// TIA Portal project "maqueta brazo" (V15)
// Vorlageprojekt für das Buch mit Zielsystem S7-1200

(* hardware
DEVICE "S7-1200-Station_1"  S7-1200 Station
   slot 0: "Baugruppenträger_0"  Rack  V1.0
   slot 1: "PLC_1"  CPU 1211C DC/DC/DC  6ES7 211-1AE40-0XB0  V4.1
*)

// ===== PLC "PLC_1"  CPU 1211C DC/DC/DC =====

VAR_GLOBAL   // PLC tag table "Standard-Variablentabelle"
   "conteo para desactivar seta" AT %MW300 : Int;
   "motor derecha" AT %Q0.4 : Bool;   // motor brazo
   "Tag_1" AT %M11.7 : Bool;
   "sensor brazo bajado_m" AT %M12.0 : Bool;
   "Step_6" AT %M12.1 : Bool;
   "conteo Z" AT %MW305 : Int;
   "Tag_2" AT %M100.5 : Bool;
   "Tag_4" AT %M150.0 : Bool;
   "conteo Y" AT %MW310 : Int;
   "brazo arriba" AT %M12.2 : Bool;
   "resto_Z" AT %MW315 : Int;
   "brazo en reposo" AT %M12.3 : Bool;
   "brazo a la derecha" AT %M12.4 : Bool;
   "brazo a la izquierda" AT %M12.5 : Bool;
   "Tag_3" AT %M106.0 : Bool;
END_VAR

VAR_GLOBAL   // PLC tag table "Tabla de variables estándar"
   "start_m" AT %M10.0 : Bool;   // Start pushbutton
   "stop_m" AT %M10.1 : Bool;   // Stop pushbutton
   "auto_man_m" AT %M10.2 : Bool;   // Auto/Manual selector
   "reset_m" AT %M10.3 : Bool;   // Reset pushbutton
   "a_0_m" AT %M10.4 : Bool;   // Eject cylinder backward
   "a_1_m" AT %M10.5 : Bool;   // Eject cylinder forward
   "b_0_m" AT %M10.6 : Bool;   // Blocking cylinder backward
   "b_1_m" AT %M10.7 : Bool;   // Blocking cylinder forward
   "Block_m" AT %M11.0 : Bool;   // Block presence
   "ALARM" AT %Q0.7 : Bool;   // Alarm lamp
   "Motor izquierda" AT %Q0.3 : Bool;   // Start conveyor / Motor brazo
   "ventosa" AT %Q0.0 : Bool;   // Eject cylinder forwards / el succionador activado
   "bajar brazo" AT %Q0.1 : Bool;   // Eject cylinder downwards / baja o sube brazo
   "B+" AT %Q0.2 : Bool;   // Blocking cylinder forwards / Este va a ser el cilindro
   "Step_0" AT %M400.0 : Bool;   // First step of grafcet
   "Step_1" AT %M400.1 : Bool;   // Feeding cylinder forwards
   "Step_2" AT %M400.2 : Bool;   // Verification cylinder downwards
   "Step_3" AT %M400.3 : Bool;   // Verification cylinder upwards
   "Step_4" AT %M400.4 : Bool;   // Feeding cylinder backwards
   "Step_5" AT %M400.5 : Bool;   // Body transfer cylinder forwards
   "ic" AT %M200.0 : Bool;   // Initial conditions
   "continue" AT %M200.1 : Bool;   // Go on with the Grafcet
   "body_ok" AT %M200.2 : Bool;   // Body in right position
   "start_stop_mode" AT %M200.3 : Bool;   // Auto / Manual mode of the station
   "no_air_pressure" AT %M200.4 : Bool;   // Station without air pressure
   "cycle" AT %M200.5 : Bool;   // Process cycle not finished
   "end_cycle" AT %M200.6 : Bool;   // Station 1 end cycle
   "FAS201_on_202" AT %Q200.0 : Bool;   // Fas-201 on for fas-202
   "FAS201_end_202" AT %Q200.1 : Bool;   // Process cycle finished at fas-201 for fas-202
   "FAS201_wrong_202" AT %Q200.2 : Bool;   // Body wrongly positioned for fas-202
   "FAS201_c1_202" AT %Q200.3 : Bool;   // Transfer cylinder forward for fas-202
   "Cell_1_ppA" AT %I200.4 : Bool;   // Palet presence fas-202
   "Cell_1_b0A" AT %I200.5 : Bool;   // Palet code bit 0 fas-202
   "Cell_1_b1A" AT %I200.6 : Bool;   // Palet code bit 1 fas-202
   "Cell_1_b2A" AT %I200.7 : Bool;   // Palet code bit 2 fas-202
   "First_SC" AT %M3.6 : Bool;
   "Tag_21" AT %M201.7 : Bool;
   "Tag_6" AT %M100.4 : Bool;
   "Cell_1_on" AT %I200.0 : Bool;   // Fas-202 on
   "Cell_1_end" AT %I200.1 : Bool;   // Cycle finished at fas-202
   "Cell_1_busy" AT %I200.2 : Bool;   // Fas-202 busy
   "Cell_1_alarm" AT %I200.3 : Bool;
   "sensor_start" AT %I1.1 : Bool;   // Capacitive sensor start conveyor
   "sensor_end" AT %I1.2 : Bool;   // Capacitive sensor end conveyor
   "brazo en movimiento" AT %I1.0 : Bool;   // Detected white block / brazo eje horizontal
   "System_Byte" AT %MB254 : Byte;
   "FirstScan" AT %M254.0 : Bool;
   "DiagStatusUpdate" AT %M254.1 : Bool;
   "AlwaysTRUE" AT %M254.2 : Bool;
   "AlwaysFALSE" AT %M254.3 : Bool;
   "start" AT %I0.2 : Bool;   // Start pushbutton
   "stop" AT %I0.1 : Bool;   // Stop pushbutton
   "auto_man" AT %I0.3 : Bool;   // Auto/Manual selector
   "reset" AT %I0.0 : Bool;   // Reset pushbutton
   "ventosa activada" AT %I0.4 : Bool;   // Eject cylinder backward / Ventosa
   "sensor pieza" AT %I0.5 : Bool;   // Eject cylinder forward / Botón para verificar si hay pieza
   "b_0" AT %I0.6 : Bool;   // Blocking cylinder backward / cilindro detrás
   "b_1" AT %I0.7 : Bool;   // Blocking cylinder forward / cilindro delante
   "Sensor brazo bajado" AT %I1.3 : Bool;   // Block presence / Sensor que indica si el brazo está bajando o subiendo
   "Sensor_start_m" AT %M11.1 : Bool;
   "sensor_end_m" AT %M11.2 : Bool;
   "brazo en movimiento _m" AT %M11.3 : Bool;
   "Pieza a la espera" AT %M11.4 : Bool;   // Se activa cuando hay una pieza en la cinta
   "pieza cogida" AT %M11.5 : Bool;   // Se activa cuando detecta que la pieza es blanca / variable que nos indica si el brazo ha cogido la pieza
   "Piezas" AT %M11.6 : Bool;   // Cuenta el número de piezas
   "reinicio" AT %M400.6 : Bool;
END_VAR

VAR_GLOBAL CONSTANT   // PLC tag table "Tabla de variables estándar"
   "Local~AI2_1" : Hw_SubModule := 264;
   "Local~DI14_DQ10_1" : Hw_SubModule := 265;
   "OB_Main(1)" : OB_PCYCLE := 1;
   "OB_Diagnostic error interrupt" : OB_DIAG := 82;
   "None" : Pip := 65535;
   "Automatic update" : Pip := 0;
   "PIP 1" : Pip := 1;
   "PIP 2" : Pip := 2;
   "PIP 3" : Pip := 3;
   "PIP 4" : Pip := 4;
   "PIP OB Servo" : Pip := 32768;
   "Local~Interfaz_PROFINET_1~IODevice" : Hw_Device := 271;
   "Local~Interfaz_PROFINET_1~Transfer_area_1" : Hw_SubModule := 273;
   "Local~Interfaz_PROFINET_1~Transfer_area_2" : Hw_SubModule := 274;
   "Local~Exec(1)" : Hw_SubModule := 52;
   "Local(1)" : Hw_SubModule := 49;
   "Local~Interfaz_PROFINET_1~Puerto_1" : Hw_Interface := 65;
   "Local~MC(1)" : Hw_SubModule := 51;
   "Local~Common(1)" : Hw_SubModule := 50;
   "Local~Device(1)" : Hw_Device := 32;
   "Local~Configuration(1)" : Hw_SubModule := 33;
   "Local~HSC_1(1)" : Hw_Hsc := 258;
   "Local~HSC_2(1)" : Hw_Hsc := 259;
   "Local~HSC_3(1)" : Hw_Hsc := 260;
   "Local~HSC_4(1)" : Hw_Hsc := 261;
   "Local~HSC_5(1)" : Hw_Hsc := 262;
   "Local~HSC_6(1)" : Hw_Hsc := 263;
   "Local~Pulse_1(1)" : Hw_Pwm := 266;
   "Local~Pulse_2(1)" : Hw_Pwm := 267;
   "Local~Pulse_3(1)" : Hw_Pwm := 269;
   "Local~Pulse_4(1)" : Hw_Pwm := 270;
   "Local~Interfaz_PROFINET_1" : Hw_Interface := 64;
   "Local~AQ_2x14BIT_1" : Hw_SubModule := 275;
   "Local~DQ_4x24VDC_1" : Hw_SubModule := 276;
   "OB_Startup" : OB_STARTUP := 100;
END_VAR

// folder: System blocks/Program resources

DATA_BLOCK "TIMER_1"   // DB1
{ S7_Optimized_Access := 'TRUE' }
AUTHOR : Simatic
FAMILY : IEC
NAME : IEC_TMR
VERSION : 1.0
// stored: InstanceOfName IEC_TIMER
"IEC_TIMER"
BEGIN
END_DATA_BLOCK

DATA_BLOCK "TIMER_2"   // DB2
{ S7_Optimized_Access := 'TRUE' }
AUTHOR : Simatic
FAMILY : IEC
NAME : IEC_TMR
VERSION : 1.0
// stored: InstanceOfName IEC_TIMER
"IEC_TIMER"
BEGIN
END_DATA_BLOCK

DATA_BLOCK "TIMER_3"   // DB3
{ S7_Optimized_Access := 'TRUE' }
AUTHOR : Simatic
FAMILY : IEC
NAME : IEC_TMR
VERSION : 1.0
// stored: InstanceOfName IEC_TIMER
"IEC_TIMER"
BEGIN
END_DATA_BLOCK

DATA_BLOCK "IEC_Counter_0_DB"   // DB4
{ S7_Optimized_Access := 'TRUE' }
AUTHOR : Simatic
FAMILY : IEC
NAME : CNTR
VERSION : 1.0
// stored: InstanceOfName IEC_COUNTER
"IEC_COUNTER"
BEGIN
END_DATA_BLOCK

DATA_BLOCK "TIMER_6"   // DB5
{ S7_Optimized_Access := 'TRUE' }
AUTHOR : Simatic
FAMILY : IEC
NAME : IEC_TMR
VERSION : 1.0
// stored: InstanceOfName IEC_TIMER
"IEC_TIMER"
BEGIN
END_DATA_BLOCK

DATA_BLOCK "TIMER_8"   // DB6
{ S7_Optimized_Access := 'TRUE' }
AUTHOR : Simatic
FAMILY : IEC
NAME : IEC_TMR
VERSION : 1.0
// stored: InstanceOfName IEC_TIMER
"IEC_TIMER"
BEGIN
END_DATA_BLOCK

DATA_BLOCK "IEC_Timer_0_DB_3"   // DB7
{ S7_Optimized_Access := 'TRUE' }
AUTHOR : Simatic
FAMILY : IEC
NAME : IEC_TMR
VERSION : 1.0
// stored: InstanceOfName IEC_TIMER
"IEC_TIMER"
BEGIN
END_DATA_BLOCK

DATA_BLOCK "IEC_Timer_0_DB"   // DB8
{ S7_Optimized_Access := 'TRUE' }
AUTHOR : Simatic
FAMILY : IEC
NAME : IEC_TMR
VERSION : 1.0
// stored: InstanceOfName IEC_TIMER
"IEC_TIMER"
BEGIN
END_DATA_BLOCK

DATA_BLOCK "IEC_Timer_0_DB_1"   // DB9
{ S7_Optimized_Access := 'TRUE' }
AUTHOR : Simatic
FAMILY : IEC
NAME : IEC_TMR
VERSION : 1.0
// stored: InstanceOfName IEC_TIMER
"IEC_TIMER"
BEGIN
END_DATA_BLOCK

DATA_BLOCK "IEC_Counter_0_DB_2"   // DB10
{ S7_Optimized_Access := 'TRUE' }
AUTHOR : Simatic
FAMILY : IEC
NAME : CNTR
VERSION : 1.0
// stored: InstanceOfName IEC_COUNTER
"IEC_COUNTER"
BEGIN
END_DATA_BLOCK

DATA_BLOCK "IEC_Timer_0_DB_4"   // DB11
{ S7_Optimized_Access := 'TRUE' }
AUTHOR : Simatic
FAMILY : IEC
NAME : IEC_TMR
VERSION : 1.0
// stored: InstanceOfName IEC_TIMER
"IEC_TIMER"
BEGIN
END_DATA_BLOCK

DATA_BLOCK "IEC_Counter_0_DB_3"   // DB12
{ S7_Optimized_Access := 'TRUE' }
AUTHOR : Simatic
FAMILY : IEC
NAME : CNTR
VERSION : 1.0
// stored: InstanceOfName IEC_COUNTER
"IEC_COUNTER"
BEGIN
END_DATA_BLOCK

DATA_BLOCK "IEC_Timer_0_DB_2"   // DB13
{ S7_Optimized_Access := 'TRUE' }
AUTHOR : Simatic
FAMILY : IEC
NAME : IEC_TMR
VERSION : 1.0
// stored: InstanceOfName IEC_TIMER
"IEC_TIMER"
BEGIN
END_DATA_BLOCK

DATA_BLOCK "IEC_Timer_0_DB_5"   // DB14
{ S7_Optimized_Access := 'TRUE' }
AUTHOR : Simatic
FAMILY : IEC
NAME : IEC_TMR
VERSION : 1.0
// stored: InstanceOfName IEC_TIMER
"IEC_TIMER"
BEGIN
END_DATA_BLOCK

DATA_BLOCK "IEC_Timer_0_DB_7"   // DB16
{ S7_Optimized_Access := 'TRUE' }
AUTHOR : Simatic
FAMILY : IEC
NAME : IEC_TMR
VERSION : 1.0
// stored: InstanceOfName IEC_TIMER
"IEC_TIMER"
BEGIN
END_DATA_BLOCK

// folder: (top level)

FUNCTION "STEPS" : Void   // FC1, LAD
TITLE = STEPS
{ S7_Optimized_Access := 'TRUE' }
VERSION : 0.1
   VAR_TEMP   // added for the SCL form of the ladder/FBD networks
      _w1 : Bool;
   END_VAR
BEGIN

REGION Network 1: STEP 0 / Reposo
   // FIRST STEP OF GRAFCET / Para entrar a este estado, el brazo ha de estar en su posición inicial, con el brazo arriba y en posición de reposo.
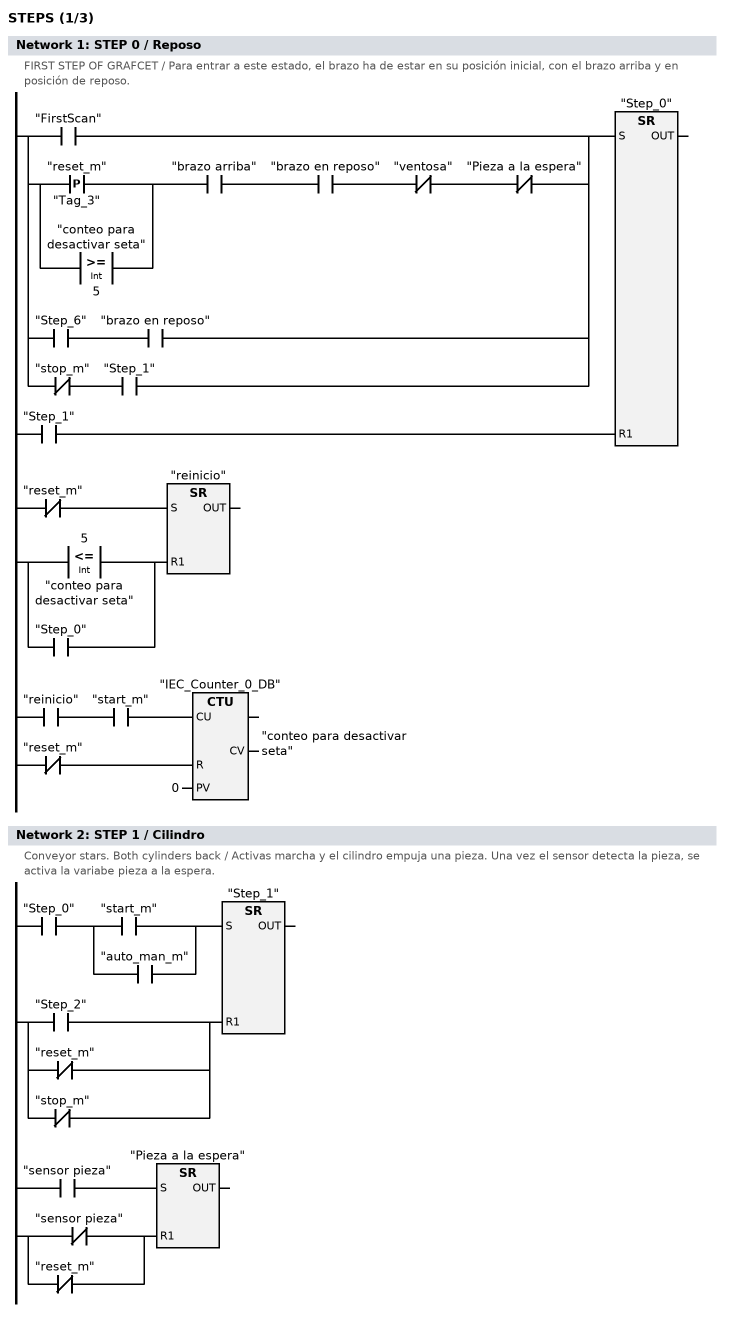
   #_w1 := "reset_m" AND NOT "Tag_3";   // rising edge of "reset_m"
   "Tag_3" := "reset_m";
   IF "FirstScan" OR ((#_w1 OR ("conteo para desactivar seta" >= 5)) AND "brazo arriba" AND "brazo en reposo" AND NOT "ventosa" AND NOT "Pieza a la espera") OR ("Step_6" AND "brazo en reposo") OR (NOT "stop_m" AND "Step_1") THEN
       "Step_0" := TRUE;   // SR flip-flop
   END_IF;
   IF "Step_1" THEN "Step_0" := FALSE; END_IF;
   IF NOT "reset_m" THEN
       "reinicio" := TRUE;   // SR flip-flop
   END_IF;
   IF (5 <= "conteo para desactivar seta") OR "Step_0" THEN "reinicio" := FALSE; END_IF;
   "IEC_Counter_0_DB".CTU(CU := "reinicio" AND "start_m",
                          R := NOT "reset_m",
                          PV := 0,
                          CV => "conteo para desactivar seta");
END_REGION

REGION Network 2: STEP 1 / Cilindro
   // Conveyor stars. Both cylinders back / Activas marcha y el cilindro empuja una pieza. Una vez el sensor detecta la pieza, se activa la variabe pieza a la espera.
   RUNG wire#powerrail
      Contact( "Step_0" )
      wire#w1
      Contact( "start_m" )
      wire#w2
      S_SR(operand := "Step_1", r1 := wire#w3)
   END_RUNG
   RUNG wire#w1
      Contact( "auto_man_m" )
   END_RUNG wire#w2
   RUNG wire#powerrail
      Contact( "Step_2" )
   END_RUNG wire#w3
   RUNG wire#powerrail
      I_Contact( "reset_m" )
   END_RUNG wire#w3
   RUNG wire#powerrail
      I_Contact( "stop_m" )
   END_RUNG wire#w3
   RUNG wire#powerrail
      Contact( "sensor pieza" )
      S_SR(operand := "Pieza a la espera", r1 := wire#w4)
   END_RUNG
   RUNG wire#powerrail
      I_Contact( "sensor pieza" )
   END_RUNG wire#w4
   RUNG wire#powerrail
      I_Contact( "reset_m" )
   END_RUNG wire#w4
   // the same network as SCL:
   IF "Step_0" AND ("start_m" OR "auto_man_m") THEN
       "Step_1" := TRUE;   // SR flip-flop
   END_IF;
   IF "Step_2" OR NOT "reset_m" OR NOT "stop_m" THEN "Step_1" := FALSE; END_IF;
   IF "sensor pieza" THEN
       "Pieza a la espera" := TRUE;   // SR flip-flop
   END_IF;
   IF NOT "sensor pieza" OR NOT "reset_m" THEN "Pieza a la espera" := FALSE; END_IF;
END_REGION

REGION Network 3: STEP 2 / movimiento brazo
   // Block the body / una vez detectado que hay pieza, el brazo deja su posición de reposo y hace un movimiento a la derecha para posicionarse encima de la pieza.
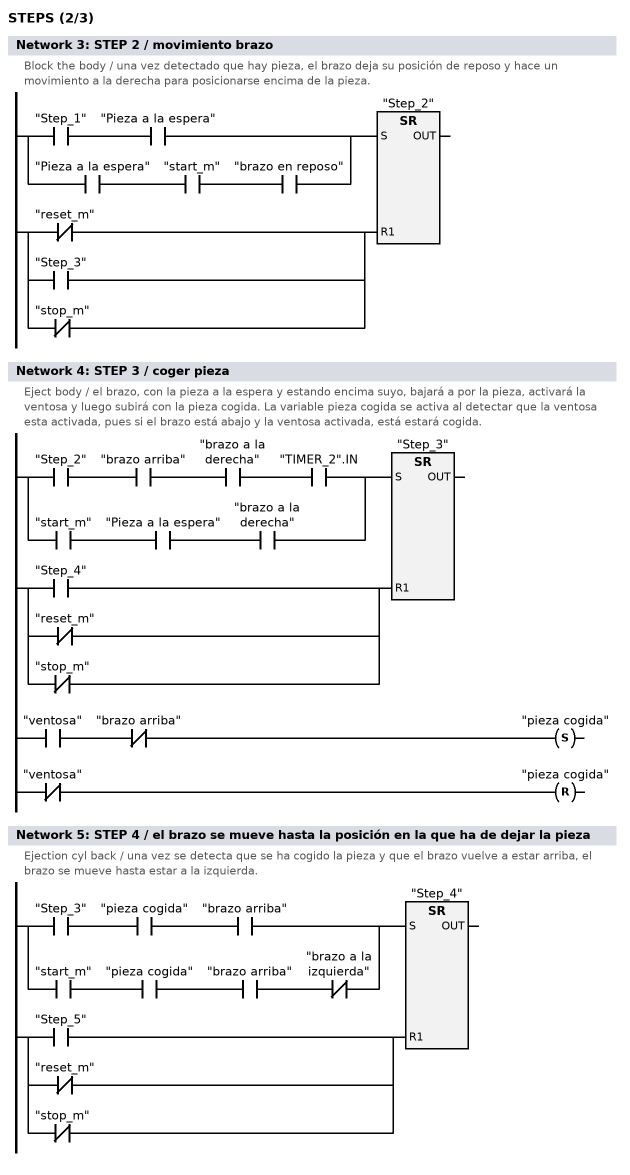
   RUNG wire#powerrail
      Contact( "Step_1" )
      Contact( "Pieza a la espera" )
      wire#w1
      S_SR(operand := "Step_2", r1 := wire#w2)
   END_RUNG
   RUNG wire#powerrail
      Contact( "Pieza a la espera" )
      Contact( "start_m" )
      Contact( "brazo en reposo" )
   END_RUNG wire#w1
   RUNG wire#powerrail
      I_Contact( "reset_m" )
   END_RUNG wire#w2
   RUNG wire#powerrail
      Contact( "Step_3" )
   END_RUNG wire#w2
   RUNG wire#powerrail
      I_Contact( "stop_m" )
   END_RUNG wire#w2
   // the same network as SCL:
   IF ("Step_1" AND "Pieza a la espera") OR ("Pieza a la espera" AND "start_m" AND "brazo en reposo") THEN
       "Step_2" := TRUE;   // SR flip-flop
   END_IF;
   IF NOT "reset_m" OR "Step_3" OR NOT "stop_m" THEN "Step_2" := FALSE; END_IF;
END_REGION

REGION Network 4: STEP 3 / coger pieza
   // Eject body / el brazo, con la pieza a la espera y estando encima suyo, bajará a por la pieza, activará la ventosa y luego subirá con la pieza cogida. La variable pieza cogida se activa al detectar que la ventosa esta activada, pues si el brazo está abajo y la ventosa activada, está estará cogida.
   RUNG wire#powerrail
      Contact( "Step_2" )
      Contact( "brazo arriba" )
      Contact( "brazo a la derecha" )
      Contact( "TIMER_2".IN )
      wire#w1
      S_SR(operand := "Step_3", r1 := wire#w2)
   END_RUNG
   RUNG wire#powerrail
      Contact( "start_m" )
      Contact( "Pieza a la espera" )
      Contact( "brazo a la derecha" )
   END_RUNG wire#w1
   RUNG wire#powerrail
      Contact( "Step_4" )
   END_RUNG wire#w2
   RUNG wire#powerrail
      I_Contact( "reset_m" )
   END_RUNG wire#w2
   RUNG wire#powerrail
      I_Contact( "stop_m" )
   END_RUNG wire#w2
   RUNG wire#powerrail
      Contact( "ventosa" )
      I_Contact( "brazo arriba" )
      S_Coil( "pieza cogida" )
   END_RUNG
   RUNG wire#powerrail
      I_Contact( "ventosa" )
      R_Coil( "pieza cogida" )
   END_RUNG
   // the same network as SCL:
   IF ("Step_2" AND "brazo arriba" AND "brazo a la derecha" AND "TIMER_2".IN) OR ("start_m" AND "Pieza a la espera" AND "brazo a la derecha") THEN
       "Step_3" := TRUE;   // SR flip-flop
   END_IF;
   IF "Step_4" OR NOT "reset_m" OR NOT "stop_m" THEN "Step_3" := FALSE; END_IF;
   IF "ventosa" AND NOT "brazo arriba" THEN "pieza cogida" := TRUE; END_IF;
   IF NOT "ventosa" THEN "pieza cogida" := FALSE; END_IF;
END_REGION

REGION Network 5: STEP 4 / el brazo se mueve hasta la posición en la que ha de dejar la pieza
   // Ejection cyl back / una vez se detecta que se ha cogido la pieza y que el brazo vuelve a estar arriba, el brazo se mueve hasta estar a la izquierda.
   RUNG wire#powerrail
      Contact( "Step_3" )
      Contact( "pieza cogida" )
      Contact( "brazo arriba" )
      wire#w1
      S_SR(operand := "Step_4", r1 := wire#w2)
   END_RUNG
   RUNG wire#powerrail
      Contact( "start_m" )
      Contact( "pieza cogida" )
      Contact( "brazo arriba" )
      I_Contact( "brazo a la izquierda" )
   END_RUNG wire#w1
   RUNG wire#powerrail
      Contact( "Step_5" )
   END_RUNG wire#w2
   RUNG wire#powerrail
      I_Contact( "reset_m" )
   END_RUNG wire#w2
   RUNG wire#powerrail
      I_Contact( "stop_m" )
   END_RUNG wire#w2
   // the same network as SCL:
   IF ("Step_3" AND "pieza cogida" AND "brazo arriba") OR ("start_m" AND "pieza cogida" AND "brazo arriba" AND NOT "brazo a la izquierda") THEN
       "Step_4" := TRUE;   // SR flip-flop
   END_IF;
   IF "Step_5" OR NOT "reset_m" OR NOT "stop_m" THEN "Step_4" := FALSE; END_IF;
END_REGION

REGION Network 6: dejar pieza
   // una vez detecta que la pieza está a la izquierda, con la pieza cogida, bajará el brazo para dejar la pieza.
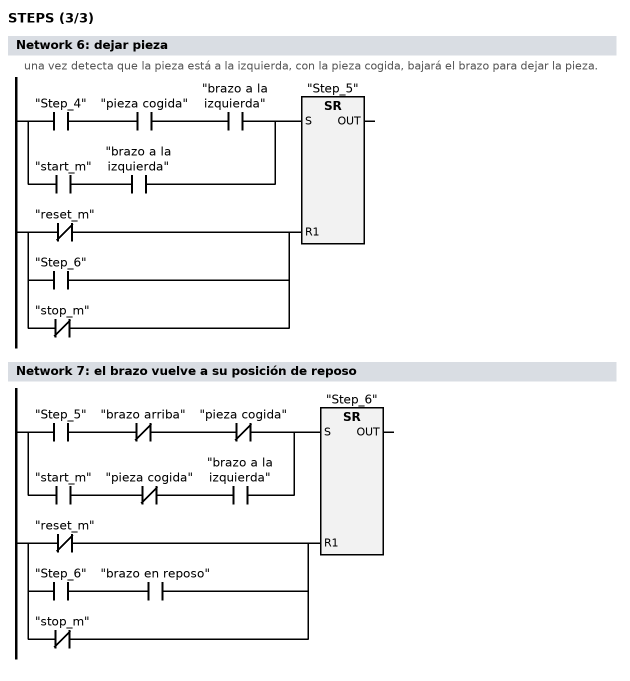
   RUNG wire#powerrail
      Contact( "Step_4" )
      Contact( "pieza cogida" )
      Contact( "brazo a la izquierda" )
      wire#w1
      S_SR(operand := "Step_5", r1 := wire#w2)
   END_RUNG
   RUNG wire#powerrail
      Contact( "start_m" )
      Contact( "brazo a la izquierda" )
   END_RUNG wire#w1
   RUNG wire#powerrail
      I_Contact( "reset_m" )
   END_RUNG wire#w2
   RUNG wire#powerrail
      Contact( "Step_6" )
   END_RUNG wire#w2
   RUNG wire#powerrail
      I_Contact( "stop_m" )
   END_RUNG wire#w2
   // the same network as SCL:
   IF ("Step_4" AND "pieza cogida" AND "brazo a la izquierda") OR ("start_m" AND "brazo a la izquierda") THEN
       "Step_5" := TRUE;   // SR flip-flop
   END_IF;
   IF NOT "reset_m" OR "Step_6" OR NOT "stop_m" THEN "Step_5" := FALSE; END_IF;
END_REGION

REGION Network 7: el brazo vuelve a su posición de reposo
   RUNG wire#powerrail
      Contact( "Step_5" )
      I_Contact( "brazo arriba" )
      I_Contact( "pieza cogida" )
      wire#w1
      S_SR(operand := "Step_6", r1 := wire#w2)
   END_RUNG
   RUNG wire#powerrail
      Contact( "start_m" )
      I_Contact( "pieza cogida" )
      Contact( "brazo a la izquierda" )
   END_RUNG wire#w1
   RUNG wire#powerrail
      I_Contact( "reset_m" )
   END_RUNG wire#w2
   RUNG wire#powerrail
      Contact( "Step_6" )
      Contact( "brazo en reposo" )
   END_RUNG wire#w2
   RUNG wire#powerrail
      I_Contact( "stop_m" )
   END_RUNG wire#w2
   // the same network as SCL:
   #_w1 := NOT "reset_m" OR ("Step_6" AND "brazo en reposo") OR NOT "stop_m";
   IF ("Step_5" AND NOT "brazo arriba" AND NOT "pieza cogida") OR ("start_m" AND NOT "pieza cogida" AND "brazo a la izquierda") THEN
       "Step_6" := TRUE;   // SR flip-flop
   END_IF;
   IF #_w1 THEN "Step_6" := FALSE; END_IF;
END_REGION
END_FUNCTION

FUNCTION "TIMERS" : Void   // FC2, LAD
TITLE = TIMERS
{ S7_Optimized_Access := 'TRUE' }
VERSION : 0.1
BEGIN

REGION Network 1: TIMER 1
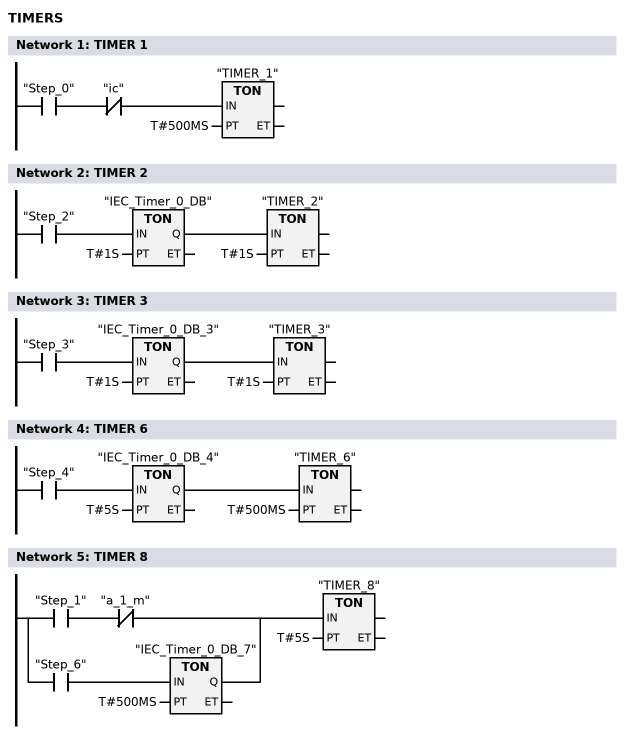
   "TIMER_1".TON(IN := "Step_0" AND NOT "ic", PT := T#500MS);
END_REGION

REGION Network 2: TIMER 2
   "IEC_Timer_0_DB".TON(IN := "Step_2", PT := T#1S);
   "TIMER_2".TON(IN := "IEC_Timer_0_DB".Q, PT := T#1S);
END_REGION

REGION Network 3: TIMER 3
   "IEC_Timer_0_DB_3".TON(IN := "Step_3", PT := T#1S);
   "TIMER_3".TON(IN := "IEC_Timer_0_DB_3".Q, PT := T#1S);
END_REGION

REGION Network 4: TIMER 6
   "IEC_Timer_0_DB_4".TON(IN := "Step_4", PT := T#5S);
   "TIMER_6".TON(IN := "IEC_Timer_0_DB_4".Q, PT := T#500MS);
END_REGION

REGION Network 5: TIMER 8
   "IEC_Timer_0_DB_7".TON(IN := "Step_6", PT := T#500MS);
   "TIMER_8".TON(IN := ("Step_1" AND NOT "a_1_m") OR "IEC_Timer_0_DB_7".Q, PT := T#5S);
END_REGION
END_FUNCTION

FUNCTION "WORKBITS" : Void   // FC3, LAD
TITLE = WORKBITS
{ S7_Optimized_Access := 'TRUE' }
VERSION : 0.1
BEGIN

REGION Network 1: START STOP MODE
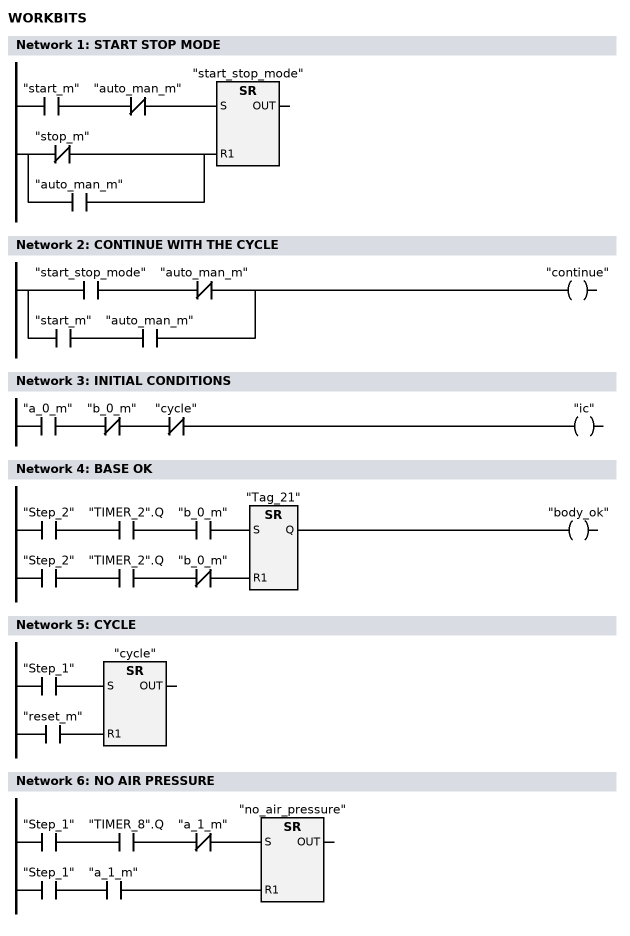
   RUNG wire#powerrail
      Contact( "start_m" )
      I_Contact( "auto_man_m" )
      S_SR(operand := "start_stop_mode", r1 := wire#w1)
   END_RUNG
   RUNG wire#powerrail
      I_Contact( "stop_m" )
   END_RUNG wire#w1
   RUNG wire#powerrail
      Contact( "auto_man_m" )
   END_RUNG wire#w1
   // the same network as SCL:
   IF "start_m" AND NOT "auto_man_m" THEN
       "start_stop_mode" := TRUE;   // SR flip-flop
   END_IF;
   IF NOT "stop_m" OR "auto_man_m" THEN "start_stop_mode" := FALSE; END_IF;
END_REGION

REGION Network 2: CONTINUE WITH THE CYCLE
   RUNG wire#powerrail
      Contact( "start_stop_mode" )
      I_Contact( "auto_man_m" )
      wire#w1
      Coil( "continue" )
   END_RUNG
   RUNG wire#powerrail
      Contact( "start_m" )
      Contact( "auto_man_m" )
   END_RUNG wire#w1
   // the same network as SCL:
   "continue" := ("start_stop_mode" AND NOT "auto_man_m") OR ("start_m" AND "auto_man_m");
END_REGION

REGION Network 3: INITIAL CONDITIONS
   RUNG wire#powerrail
      Contact( "a_0_m" )
      I_Contact( "b_0_m" )
      I_Contact( "cycle" )
      Coil( "ic" )
   END_RUNG
   // the same network as SCL:
   "ic" := "a_0_m" AND NOT "b_0_m" AND NOT "cycle";
END_REGION

REGION Network 4: BASE OK
   RUNG wire#powerrail
      Contact( "Step_2" )
      Contact( "TIMER_2".Q )
      Contact( "b_0_m" )
      S_SR(operand := "Tag_21", r1 := wire#w1)
      Coil( "body_ok" )
   END_RUNG
   RUNG wire#powerrail
      Contact( "Step_2" )
      Contact( "TIMER_2".Q )
      I_Contact( "b_0_m" )
   END_RUNG wire#w1
   // the same network as SCL:
   IF "Step_2" AND "TIMER_2".Q AND "b_0_m" THEN
       "Tag_21" := TRUE;   // SR flip-flop
   END_IF;
   IF "Step_2" AND "TIMER_2".Q AND NOT "b_0_m" THEN "Tag_21" := FALSE; END_IF;
   "body_ok" := "Tag_21";
END_REGION

REGION Network 5: CYCLE
   RUNG wire#powerrail
      Contact( "Step_1" )
      S_SR(operand := "cycle", r1 := wire#w1)
   END_RUNG
   RUNG wire#powerrail
      Contact( "reset_m" )
   END_RUNG wire#w1
   // the same network as SCL:
   IF "Step_1" THEN
       "cycle" := TRUE;   // SR flip-flop
   END_IF;
   IF "reset_m" THEN "cycle" := FALSE; END_IF;
END_REGION

REGION Network 6: NO AIR PRESSURE
   RUNG wire#powerrail
      Contact( "Step_1" )
      Contact( "TIMER_8".Q )
      I_Contact( "a_1_m" )
      S_SR(operand := "no_air_pressure", r1 := wire#w1)
   END_RUNG
   RUNG wire#powerrail
      Contact( "Step_1" )
      Contact( "a_1_m" )
   END_RUNG wire#w1
   // the same network as SCL:
   IF "Step_1" AND "TIMER_8".Q AND NOT "a_1_m" THEN
       "no_air_pressure" := TRUE;   // SR flip-flop
   END_IF;
   IF "Step_1" AND "a_1_m" THEN "no_air_pressure" := FALSE; END_IF;
END_REGION
END_FUNCTION

FUNCTION "OUTPUTS" : Void   // FC4, LAD
TITLE = OUTPUTS
{ S7_Optimized_Access := 'TRUE' }
VERSION : 0.1
BEGIN

REGION Network 1: ALARM
   // NO MATERIAL LAMP FLASHING
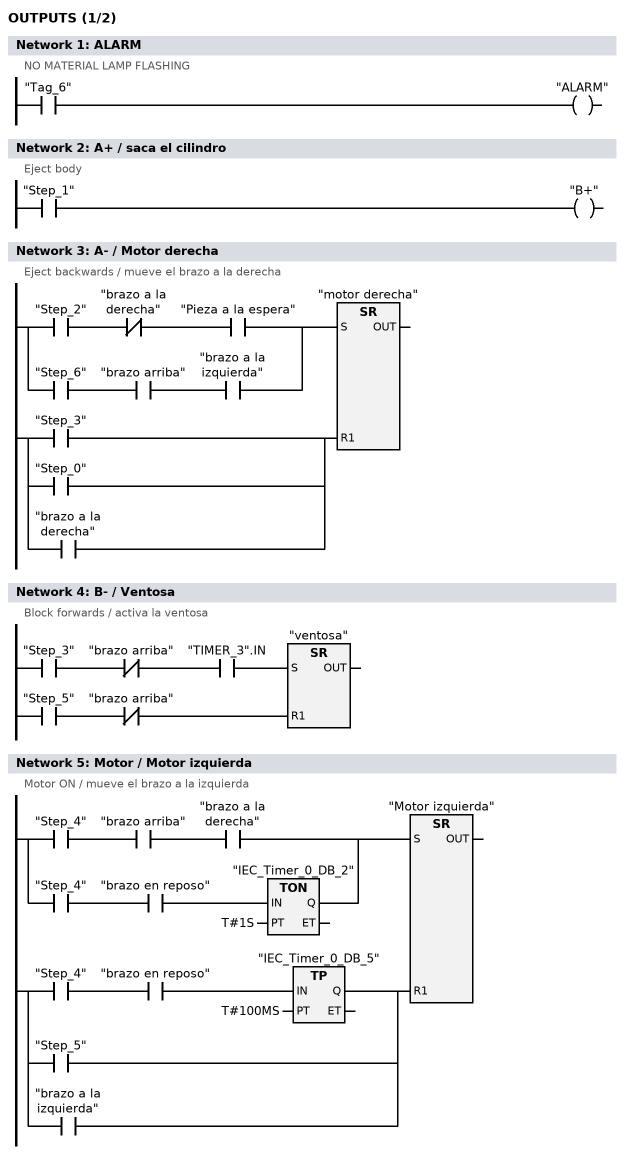
   RUNG wire#powerrail
      Contact( "Tag_6" )
      Coil( "ALARM" )
   END_RUNG
   // the same network as SCL:
   "ALARM" := "Tag_6";
END_REGION

REGION Network 2: A+ / saca el cilindro
   // Eject body
   RUNG wire#powerrail
      Contact( "Step_1" )
      Coil( "B+" )
   END_RUNG
   // the same network as SCL:
   "B+" := "Step_1";
END_REGION

REGION Network 3: A- / Motor derecha
   // Eject backwards / mueve el brazo a la derecha
   RUNG wire#powerrail
      Contact( "Step_2" )
      I_Contact( "brazo a la derecha" )
      Contact( "Pieza a la espera" )
      wire#w1
      S_SR(operand := "motor derecha", r1 := wire#w2)
   END_RUNG
   RUNG wire#powerrail
      Contact( "Step_6" )
      Contact( "brazo arriba" )
      Contact( "brazo a la izquierda" )
   END_RUNG wire#w1
   RUNG wire#powerrail
      Contact( "Step_3" )
   END_RUNG wire#w2
   RUNG wire#powerrail
      Contact( "Step_0" )
   END_RUNG wire#w2
   RUNG wire#powerrail
      Contact( "brazo a la derecha" )
   END_RUNG wire#w2
   // the same network as SCL:
   IF ("Step_2" AND NOT "brazo a la derecha" AND "Pieza a la espera") OR ("Step_6" AND "brazo arriba" AND "brazo a la izquierda") THEN
       "motor derecha" := TRUE;   // SR flip-flop
   END_IF;
   IF "Step_3" OR "Step_0" OR "brazo a la derecha" THEN "motor derecha" := FALSE; END_IF;
END_REGION

REGION Network 4: B- / Ventosa
   // Block forwards / activa la ventosa
   RUNG wire#powerrail
      Contact( "Step_3" )
      I_Contact( "brazo arriba" )
      Contact( "TIMER_3".IN )
      S_SR(operand := "ventosa", r1 := wire#w1)
   END_RUNG
   RUNG wire#powerrail
      Contact( "Step_5" )
      I_Contact( "brazo arriba" )
   END_RUNG wire#w1
   // the same network as SCL:
   IF "Step_3" AND NOT "brazo arriba" AND "TIMER_3".IN THEN
       "ventosa" := TRUE;   // SR flip-flop
   END_IF;
   IF "Step_5" AND NOT "brazo arriba" THEN "ventosa" := FALSE; END_IF;
END_REGION

REGION Network 5: Motor / Motor izquierda
   // Motor ON / mueve el brazo a la izquierda
   "IEC_Timer_0_DB_2".TON(IN := "Step_4" AND "brazo en reposo", PT := T#1S);
   "IEC_Timer_0_DB_5".TP(IN := "Step_4" AND "brazo en reposo", PT := T#100MS);
   IF ("Step_4" AND "brazo arriba" AND "brazo a la derecha") OR "IEC_Timer_0_DB_2".Q THEN
       "Motor izquierda" := TRUE;   // SR flip-flop
   END_IF;
   IF "IEC_Timer_0_DB_5".Q OR "Step_5" OR "brazo a la izquierda" THEN "Motor izquierda" := FALSE; END_IF;
END_REGION

REGION Network 6: bajar-subir brazo
   // baja el brazo
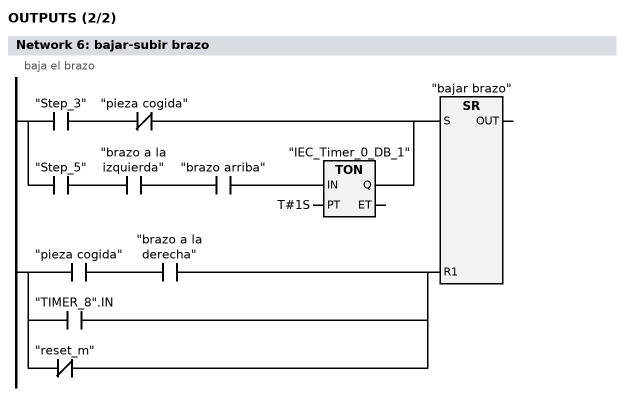
   "IEC_Timer_0_DB_1".TON(IN := "Step_5" AND "brazo a la izquierda" AND "brazo arriba", PT := T#1S);
   IF ("Step_3" AND NOT "pieza cogida") OR "IEC_Timer_0_DB_1".Q THEN
       "bajar brazo" := TRUE;   // SR flip-flop
   END_IF;
   IF ("pieza cogida" AND "brazo a la derecha") OR "TIMER_8".IN OR NOT "reset_m" THEN
       "bajar brazo" := FALSE;
   END_IF;
END_REGION
END_FUNCTION

FUNCTION "COMMS" : Void   // FC5, LAD
TITLE = PROFINET COMMUNICATION
{ S7_Optimized_Access := 'TRUE' }
VERSION : 0.1
BEGIN

REGION Network 1: FAS-201 ON FOR FAS-202
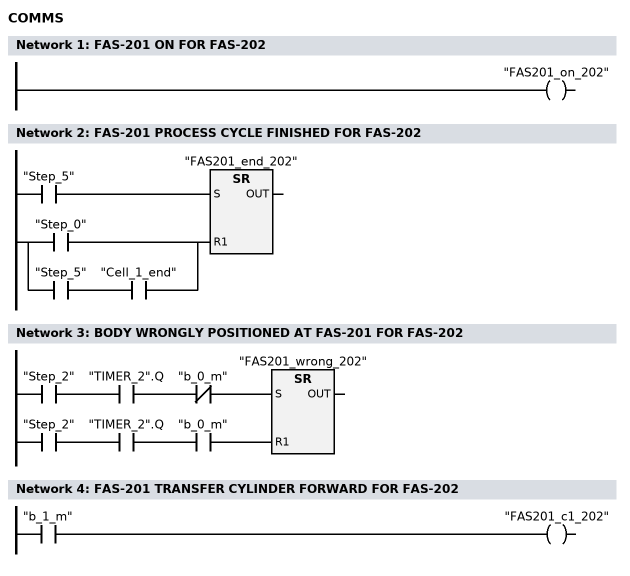
   RUNG wire#powerrail
      Coil( "FAS201_on_202" )
   END_RUNG
   // the same network as SCL:
   "FAS201_on_202" := TRUE;
END_REGION

REGION Network 2: FAS-201 PROCESS CYCLE FINISHED FOR FAS-202
   RUNG wire#powerrail
      Contact( "Step_5" )
      S_SR(operand := "FAS201_end_202", r1 := wire#w1)
   END_RUNG
   RUNG wire#powerrail
      Contact( "Step_0" )
   END_RUNG wire#w1
   RUNG wire#powerrail
      Contact( "Step_5" )
      Contact( "Cell_1_end" )
   END_RUNG wire#w1
   // the same network as SCL:
   IF "Step_5" THEN
       "FAS201_end_202" := TRUE;   // SR flip-flop
   END_IF;
   IF "Step_0" OR ("Step_5" AND "Cell_1_end") THEN "FAS201_end_202" := FALSE; END_IF;
END_REGION

REGION Network 3: BODY WRONGLY POSITIONED AT FAS-201 FOR FAS-202
   RUNG wire#powerrail
      Contact( "Step_2" )
      Contact( "TIMER_2".Q )
      I_Contact( "b_0_m" )
      S_SR(operand := "FAS201_wrong_202", r1 := wire#w1)
   END_RUNG
   RUNG wire#powerrail
      Contact( "Step_2" )
      Contact( "TIMER_2".Q )
      Contact( "b_0_m" )
   END_RUNG wire#w1
   // the same network as SCL:
   IF "Step_2" AND "TIMER_2".Q AND NOT "b_0_m" THEN
       "FAS201_wrong_202" := TRUE;   // SR flip-flop
   END_IF;
   IF "Step_2" AND "TIMER_2".Q AND "b_0_m" THEN "FAS201_wrong_202" := FALSE; END_IF;
END_REGION

REGION Network 4: FAS-201 TRANSFER CYLINDER FORWARD FOR FAS-202
   RUNG wire#powerrail
      Contact( "b_1_m" )
      Coil( "FAS201_c1_202" )
   END_RUNG
   // the same network as SCL:
   "FAS201_c1_202" := "b_1_m";
END_REGION
END_FUNCTION

FUNCTION "I_to_M" : Void   // FC6, LAD
{ S7_Optimized_Access := 'TRUE' }
VERSION : 0.1
BEGIN

REGION Network 1: Entradas Byte 0
   // El byte 0 de entradas asigna las marcas del byte 0 los a0-1 y b0-1 son las entradas de cilindro
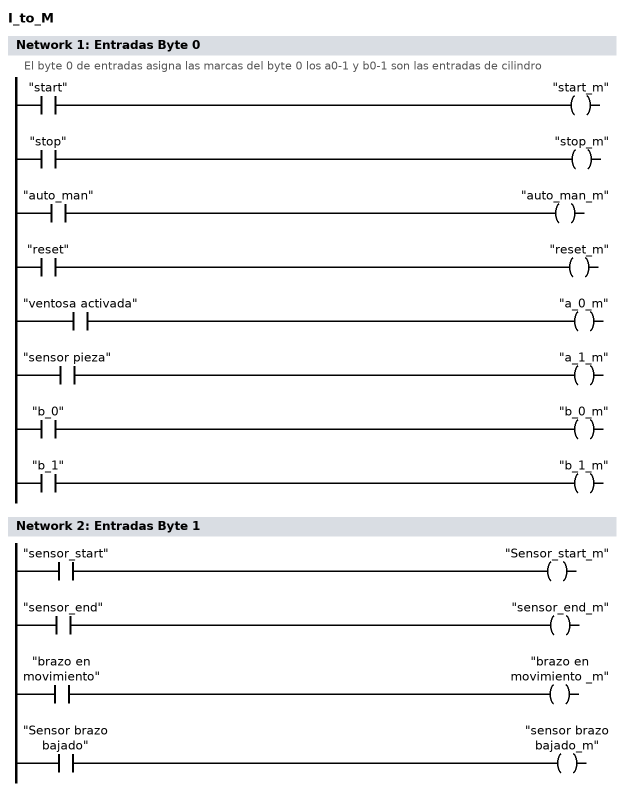
   RUNG wire#powerrail
      Contact( "start" )
      Coil( "start_m" )
   END_RUNG
   RUNG wire#powerrail
      Contact( "stop" )
      Coil( "stop_m" )
   END_RUNG
   RUNG wire#powerrail
      Contact( "auto_man" )
      Coil( "auto_man_m" )
   END_RUNG
   RUNG wire#powerrail
      Contact( "reset" )
      Coil( "reset_m" )
   END_RUNG
   RUNG wire#powerrail
      Contact( "ventosa activada" )
      Coil( "a_0_m" )
   END_RUNG
   RUNG wire#powerrail
      Contact( "sensor pieza" )
      Coil( "a_1_m" )
   END_RUNG
   RUNG wire#powerrail
      Contact( "b_0" )
      Coil( "b_0_m" )
   END_RUNG
   RUNG wire#powerrail
      Contact( "b_1" )
      Coil( "b_1_m" )
   END_RUNG
   // the same network as SCL:
   "start_m" := "start";
   "stop_m" := "stop";
   "auto_man_m" := "auto_man";
   "reset_m" := "reset";
   "a_0_m" := "ventosa activada";
   "a_1_m" := "sensor pieza";
   "b_0_m" := "b_0";
   "b_1_m" := "b_1";
END_REGION

REGION Network 2: Entradas Byte 1
   RUNG wire#powerrail
      Contact( "sensor_start" )
      Coil( "Sensor_start_m" )
   END_RUNG
   RUNG wire#powerrail
      Contact( "sensor_end" )
      Coil( "sensor_end_m" )
   END_RUNG
   RUNG wire#powerrail
      Contact( "brazo en movimiento" )
      Coil( "brazo en movimiento _m" )
   END_RUNG
   RUNG wire#powerrail
      Contact( "Sensor brazo bajado" )
      Coil( "sensor brazo bajado_m" )
   END_RUNG
   // the same network as SCL:
   "Sensor_start_m" := "sensor_start";
   "sensor_end_m" := "sensor_end";
   "brazo en movimiento _m" := "brazo en movimiento";
   "sensor brazo bajado_m" := "Sensor brazo bajado";
END_REGION
END_FUNCTION

FUNCTION "contadores" : Void   // FC7, LAD
{ S7_Optimized_Access := 'TRUE' }
VERSION : 0.1
BEGIN

REGION Network 1: conteo brazo Z
   // Cuenta cada vez que el sensor de movimiento del brazo se activa
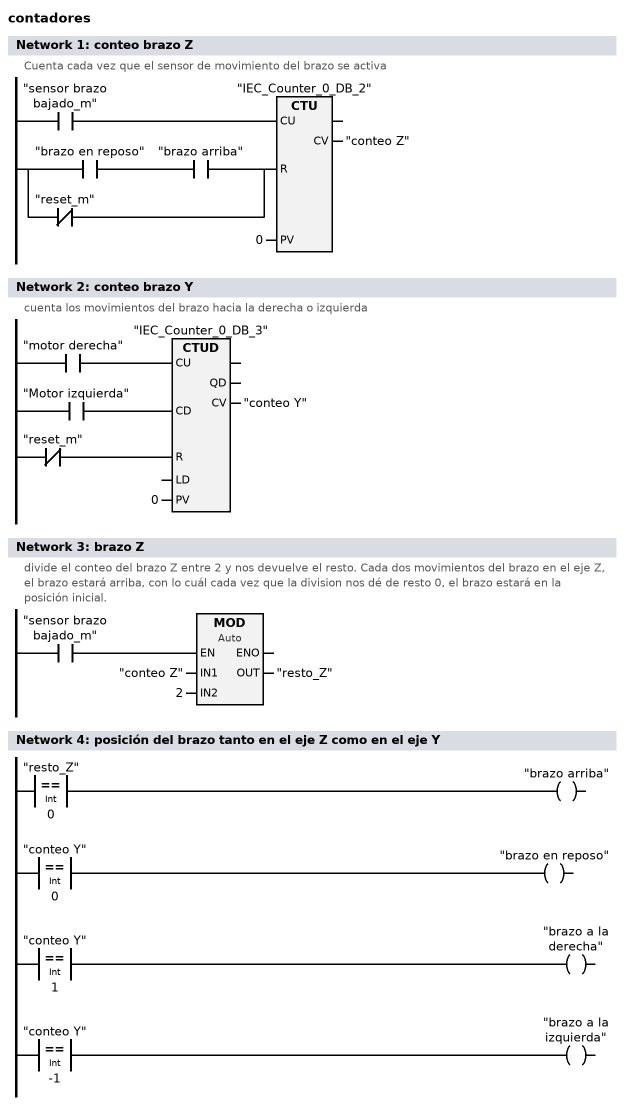
   "IEC_Counter_0_DB_2".CTU(CU := "sensor brazo bajado_m",
                           R := ("brazo en reposo" AND "brazo arriba") OR NOT "reset_m",
                           PV := 0,
                           CV => "conteo Z");
END_REGION

REGION Network 2: conteo brazo Y
   // cuenta los movimientos del brazo hacia la derecha o izquierda
   "IEC_Counter_0_DB_3".CTUD(CU := "motor derecha",
                           CD := "Motor izquierda",
                           R := NOT "reset_m",
                           PV := 0,
                           CV => "conteo Y");
END_REGION

REGION Network 3: brazo Z
   // divide el conteo del brazo Z entre 2 y nos devuelve el resto. Cada dos movimientos del brazo en el eje Z, el brazo estará arriba, con lo cuál cada vez que la division nos dé de resto 0, el brazo estará en la posición inicial.
   RUNG wire#powerrail
      Contact( "sensor brazo bajado_m" )
      Mod(in1 := "conteo Z", in2 := 2, out => "resto_Z")
   END_RUNG
   // the same network as SCL:
   IF "sensor brazo bajado_m" THEN "resto_Z" := "conteo Z" MOD 2; END_IF;
END_REGION

REGION Network 4: posición del brazo tanto en el eje Z como en el eje Y
   RUNG wire#powerrail
      { S7_Templates := "SrcType := Int" } EQ_Contact(in1 := "resto_Z", in2 := 0)
      Coil( "brazo arriba" )
   END_RUNG
   RUNG wire#powerrail
      { S7_Templates := "SrcType := Int" } EQ_Contact(in1 := "conteo Y", in2 := 0)
      Coil( "brazo en reposo" )
   END_RUNG
   RUNG wire#powerrail
      { S7_Templates := "SrcType := Int" } EQ_Contact(in1 := "conteo Y", in2 := 1)
      Coil( "brazo a la derecha" )
   END_RUNG
   RUNG wire#powerrail
      { S7_Templates := "SrcType := Int" } EQ_Contact(in1 := "conteo Y", in2 := -1)
      Coil( "brazo a la izquierda" )
   END_RUNG
   // the same network as SCL:
   "brazo arriba" := "resto_Z" = 0;
   "brazo en reposo" := "conteo Y" = 0;
   "brazo a la derecha" := "conteo Y" = 1;
   "brazo a la izquierda" := "conteo Y" = (-1);
END_REGION
END_FUNCTION

FUNCTION "MHJ-PLC-Lab-Function-S71200" : Void   // FC9000, SCL
{ S7_Optimized_Access := 'TRUE' }
VERSION : 0.1
   VAR_TEMP
      rdTimeReturn : Int;
      outputTime : DTL;
      SyncVal : Byte;
      forVal : Int;
      forVal_2 : Int;
      Value : Byte;
   END_VAR
   VAR CONSTANT
      CompVal : Byte := 16#34;
      Value_01 : Byte := 16#11;
      Value_01_DW : DWord := 16#A165_D992;
      Value_02_DW : DWord := 16#58BE_4401;
   END_VAR
BEGIN

   #Value:=PEEK(area := 16#82,
        dbNumber := 0,
        byteOffset := 511);
   #Value := #Value + 1;

   POKE(area := 16#82,
        dbNumber := 0,
        byteOffset := 511,
        value := #Value);

   POKE(area:=16#81,
        dbNumber:=0,
        byteOffset:=1016,
        value:=#Value_01_DW);
   POKE(area := 16#81,
        dbNumber := 0,
        byteOffset := 1020,
        value := #Value_02_DW);

   POKE(area := 16#81,
        dbNumber := 0,
        byteOffset := 511,
        value := B#16#00);

   FOR #forVal := 0 TO 120 DO
       FOR #forVal_2:=0 TO 10 DO
           #rdTimeReturn:=RD_SYS_T(#outputTime);
           #rdTimeReturn := WR_SYS_T(#outputTime);
           #rdTimeReturn := RD_SYS_T(#outputTime);
           #rdTimeReturn := WR_SYS_T(#outputTime);
       END_FOR;
       #SyncVal:= PEEK(area := 16#81,
                      dbNumber := 0,
                      byteOffset := 511);
       IF #SyncVal = #CompVal THEN
          GOTO M_1;
       END_IF;
   END_FOR;
   RETURN;

   M_1:
   POKE(area := 16#81,
        dbNumber := 0,
        byteOffset := 511,
        value := B#16#0);
END_FUNCTION

ORGANIZATION_BLOCK "Main"   // OB1, LAD, ProgramCycle
TITLE = "Main Program Sweep (Cycle)"
{ S7_Optimized_Access := 'TRUE' }
VERSION : 0.1
   VAR_INPUT
      Initial_Call : Bool;   // Initial call of this OB
      Remanence : Bool;   // =True, if remanent data are available
   END_VAR
BEGIN

REGION Network 1: Connection block for PLCSIM communications. Don't delete this network!
   // Im Netzwerk 1 wird der Konnektierungsbaustein für PLC-Lab aufgerufen.
   // Dieser Aufruf darf nicht entfernt werden!
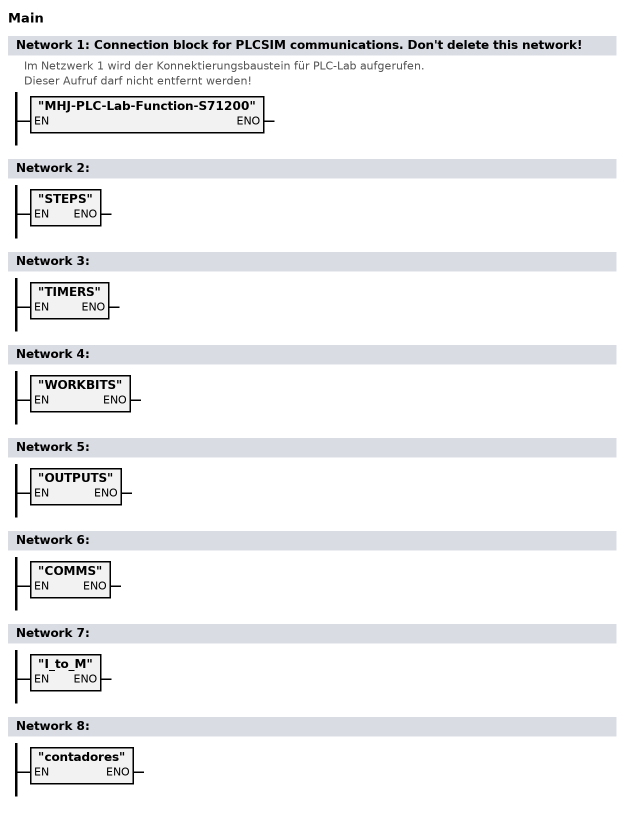
   RUNG wire#powerrail
      "MHJ-PLC-Lab-Function-S71200"()
   END_RUNG
   // the same network as SCL:
   "MHJ-PLC-Lab-Function-S71200"();
END_REGION

REGION Network 2
   RUNG wire#powerrail
      "STEPS"()
   END_RUNG
   // the same network as SCL:
   "STEPS"();
END_REGION

REGION Network 3
   RUNG wire#powerrail
      "TIMERS"()
   END_RUNG
   // the same network as SCL:
   "TIMERS"();
END_REGION

REGION Network 4
   RUNG wire#powerrail
      "WORKBITS"()
   END_RUNG
   // the same network as SCL:
   "WORKBITS"();
END_REGION

REGION Network 5
   RUNG wire#powerrail
      "OUTPUTS"()
   END_RUNG
   // the same network as SCL:
   "OUTPUTS"();
END_REGION

REGION Network 6
   RUNG wire#powerrail
      "COMMS"()
   END_RUNG
   // the same network as SCL:
   "COMMS"();
END_REGION

REGION Network 7
   RUNG wire#powerrail
      "I_to_M"()
   END_RUNG
   // the same network as SCL:
   "I_to_M"();
END_REGION

REGION Network 8
   RUNG wire#powerrail
      "contadores"()
   END_RUNG
   // the same network as SCL:
   "contadores"();
END_REGION
END_ORGANIZATION_BLOCK